// TIA Portal V18 export
ORGANIZATION_BLOCK "Main"   // OB123, LAD, ProgramCycle
TITLE = "Main Program Sweep (Cycle)"
VERSION : 0.1
// stored: AutoNumber true, IsIECCheckEnabled false, Namespace Coagulation, SetENOAutomatically false
   VAR_INPUT
      Initial_Call : Bool;   // Initial call of this OB
      Remanence : Bool;   // =True, if remanent data are available
   END_VAR
BEGIN

REGION Network 1
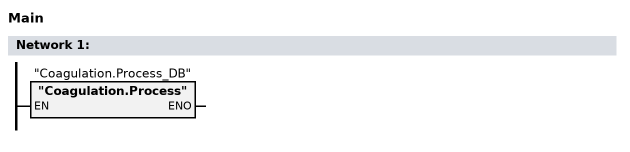
   RUNG wire#powerrail
      "Coagulation.Process_DB"()
   END_RUNG
   // the same network as SCL:
   "Coagulation.Process_DB"();   // "Coagulation.Process"
END_REGION
END_ORGANIZATION_BLOCK
